Staubli VAL3: loadCycle.pgx

public program loadCycle(string x_sItem, num& x_nResult[])
  local string l_sType
  local string l_sMessage
begin
  // load the select trajectory..already loaded
  call getTrajType(l_sType)
  if find(pt:libPath(),saveData:sPathTraj)==-1
    pt:libLoad(saveData:sPathTraj+l_sType)
    delay(0)
    if saveData:bDebug
      ? "loading JPOINT..."+saveData:sPathTraj+l_sType
    endIf
  endIf
  if isDefined(pt:tTraj[x_sItem])
    // use the type...
    sTrajCycle=x_sItem
  else
    // not FOUND
    call language:message(l_sMessage,-7)
    x_nResult=-1
    cycleStatus:bToStop=true
    popUpMsg(l_sMessage+x_sItem)
  endIf
end
